Fanuc TP program (LS listing): MAINT_ABORT.LS

/PROG  MAINT_ABORT	  Macro
/ATTR
OWNER		= MNEDITOR;
COMMENT		= "";
PROG_SIZE	= 263;
CREATE		= DATE 22-05-20  TIME 14:23:44;
MODIFIED	= DATE 22-05-20  TIME 15:27:36;
FILE_NAME	= ;
VERSION		= 0;
LINE_COUNT	= 7;
MEMORY_SIZE	= 747;
PROTECT		= READ_WRITE;
TCD:  STACK_SIZE	= 0,
      TASK_PRIORITY	= 50,
      TIME_SLICE	= 0,
      BUSY_LAMP_OFF	= 0,
      ABORT_REQUEST	= 0,
      PAUSE_REQUEST	= 0;
DEFAULT_GROUP	= 1,*,*,*,*;
CONTROL_CODE	= 00000000 00000000;
/APPL
/APPL

AUTO_SINGULARITY_HEADER;
  ENABLE_SINGULARITY_AVOIDANCE   : FALSE;
/MN
   1:  LBL[1] ;
   2:  IF (!DI[10:Manual Mode]),JMP LBL[99] ;
   3:  //CALL ABORTIT    ;
   4:  ABORT ;
   5:  LBL[99] ;
   6:  WAIT    .25(sec) ;
   7:  JMP LBL[1] ;
/POS
/END
